Fanuc KAREL source: kx00017.KL

-- PROVISIONAL review KL for V770-1; original PC SHA256 aef082953d589d07f172d8c5cb90f7959c5333146dfd0d07aa957980b7a41e44
-- Incomplete behavior may be omitted. Consult companion uncertainty JSON. Do not deploy.
PROGRAM KX00017
%NOLOCKGROUP
VAR
  I : INTEGER
  J : INTEGER
  B : BOOLEAN
  F : FILE
  S : STRING[80]
-- UNRESOLVED_DECL P type=000102
BEGIN
  -- UNRESOLVED_PC offsets 5-19; opcodes 03,2E,1B,12,13,04,14
  -- UNRESOLVED_PC offsets 24-28; opcodes 7F
END KX00017
